// Mitsubishi GX Works2 project: ServoConveyor   PLC: Q03UD

PROGRAM MAIN
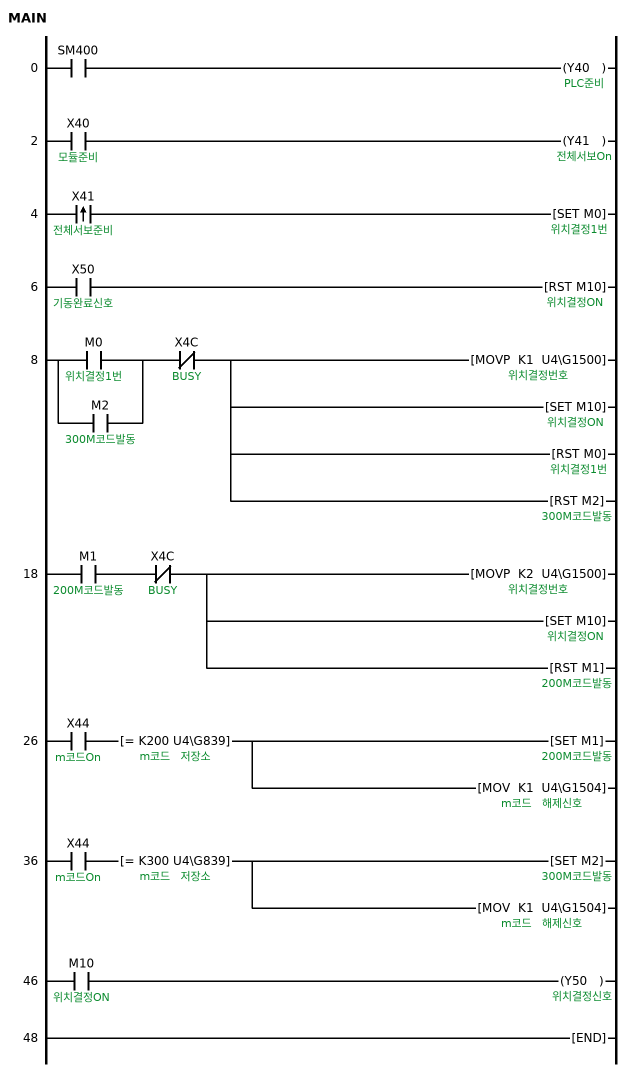
0     LD      SM400
      OUT     Y40  ; PLC준비
2     LD      X40  ; 모듈준비
      OUT     Y41  ; 전체서보On
4     LDP     X41  ; 전체서보준비
      SET     M0  ; 위치결정1번
6     LD      X50  ; 기동완료신호
      RST     M10  ; 위치결정ON
8     LD      M0  ; 위치결정1번
      OR      M2  ; 300M코드발동
      ANI     X4C  ; BUSY
      MOVP    K1 U4\G1500  ; 위치결정번호
      SET     M10  ; 위치결정ON
      RST     M0  ; 위치결정1번
      RST     M2  ; 300M코드발동
18    LD      M1  ; 200M코드발동
      ANI     X4C  ; BUSY
      MOVP    K2 U4\G1500
      SET     M10  ; 위치결정ON
      RST     M1  ; 200M코드발동
26    LD      X44  ; m코드On
      AND=    K200 U4\G839  ; m코드   저장소
      SET     M1  ; 200M코드발동
      MOV     K1 U4\G1504  ; m코드   해제신호
36    LD      X44  ; m코드On
      AND=    K300 U4\G839  ; m코드   저장소
      SET     M2  ; 300M코드발동
      MOV     K1 U4\G1504
46    LD      M10  ; 위치결정ON
      OUT     Y50  ; 위치결정신호
48    END
END_PROGRAM
